TYPE ST_ComauFeedback :
STRUCT
	q: ARRAY[0..2] OF LREAL;
	q_t: ARRAY[0..2] OF LREAL;
END_STRUCT
END_TYPE

(* stored: Version 1.1.0.1, ProductVersion 3.1.4022.7
   DUT ST_ComauFeedback: Id {48256de9-5dd0-4ad4-917f-2cc1d017818b} *)
